# EPICS autosave request: iocBoot/iocGalilTest/GALILTEST_positions.req
$(P)MTR0101.DVAL
$(P)MTR0102.DVAL
$(P)MTR0103.DVAL
$(P)MTR0104.DVAL
$(P)MTR0105.DVAL
$(P)MTR0106.DVAL
$(P)MTR0107.DVAL
$(P)MTR0108.DVAL

$(P)MTR0109.DVAL
$(P)MTR0110.DVAL
